PROGRAM MAIN
VAR
END_VAR

CONVERTERS_COMMS();

Parameters_handler();

END_PROGRAM

(* stored: Version 1.1.0.1, ProductVersion 3.1.4024.11
   POU MAIN: Id {d2dfada1-9bf9-49f9-8b63-5531027e85b3}, SpecialFunc None *)
